# EPICS IOC start-up script: iocsh/ethercatmcInt64in.iocsh
dbLoadRecords("ethercatmcInt64in.template", "P=$(P), R=$(R), ASYN_PORT=$(ASYN_PORT), DESC=$(DESC), EGU=$(EGU), ASYNADDR=$(ASYNADDR)")
